Universal Robots PolyScope program: ruch2MS333.urp

Program ruch2MS333 (installation=default directory=/programs/usbdisk createdIn=3.15.8.106339 lastSavedIn=3.15.8.106339 robotSerialNumber=2020330428)
Calibrated DH parameters: a=[0.000029, -0.241913, -0.128453, -0.000049, -0.000012, 0]; d=[0.151842, -4.082088, 33.504745, -29.309875, 0.08529, 0.082285]; alpha=[1.571059, -0.006644, 0.005794, 1.571984, -1.571997, 0]; deltaTheta=[-0.000032, 0.111537, 0.813391, -0.924919, 0.000036, 0.000016]
Robot Program (runOnlyOnce=false)
  MoveJ speed 100 deg/s, acceleration 100 deg/s^2 (useActiveTCP=true)
    Waypoint Punkt_orienta_1: TCP in base x=0.95 y=-270.681 z=692.883 mm, rx=-0.0033 ry=2.2245 rz=-2.2152 rad; joints [0.002, -89.998, 0.002, -90.001, -0.004, 0.003] deg; flange x=0.718 y=-195.682 z=693.195 mm, rx=-0.0033 ry=2.2245 rz=-2.2152 rad
    Waypoint Punkt_orienta_2: TCP in base x=-0.918 y=270.681 z=692.883 mm, rx=-1.575 ry=-0.0023 rz=0.0025 rad; joints [180, -89.996, 0.003, -90.002, -0.004, 0.005] deg; flange x=-0.689 y=195.682 z=693.195 mm, rx=-1.575 ry=-0.0023 rz=0.0025 rad
